ABB RobotStudio station: Palletixing_1.rspag

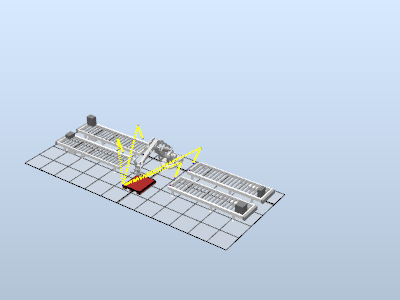
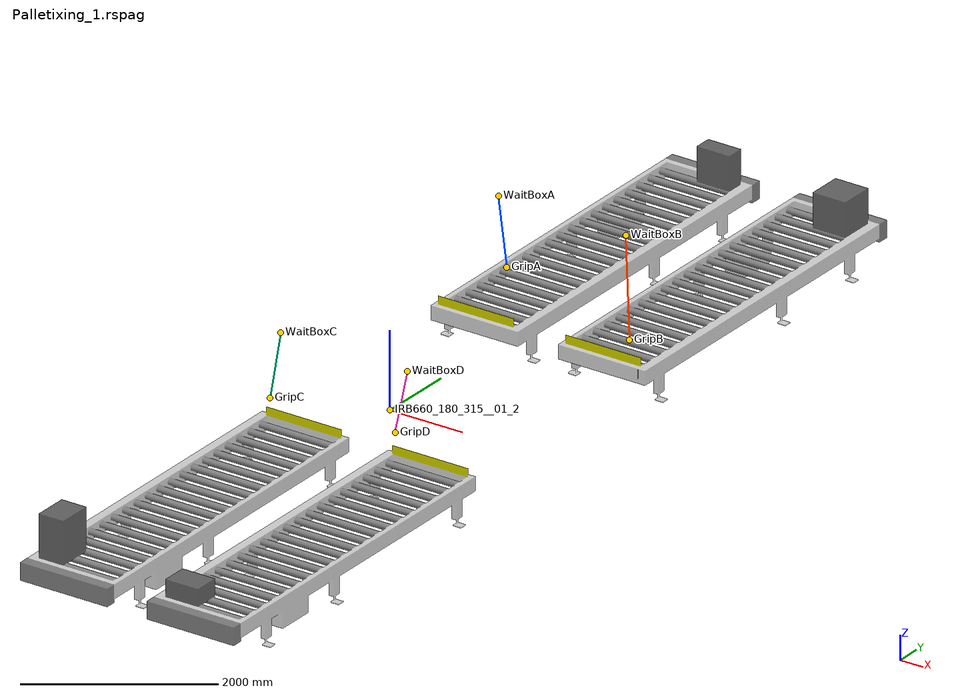
[picture v1: parts stored in the station drawn from their meshes, with robot base, taught points and paths (robot models come from the ABB library and are not in the file)]
--- station ---
Station Palletixing (saved by RobotStudio 22.3.10098.0)
Controller Controller2
  mechanical unit ROB_1: IRB660_180_315__01_2, 6 joints, base frame (0, 0, 0) mm
Layout (positions relative to the parent item):
  - IRB660_180_315__01_2 [mechanism, from Robots\IRB660_180_315__01.rslib] at (0, 0, 0) mm; joint values [0.1264, 0.8087, 0.1407, 0.1264] (rad or m)
  - Pallet1 [graphiccomponentgroup, from test\Pallet1.rslib] at (1000, 840, 377.87) mm, rotated rx 0 ry 0 rz 180 deg
    - MainBody [part, from test\Pallet1.rslib] at (-1900.1, 384.24, -377.87) mm
  - SC_InFeederA [smart component] at (435, 5540, 435) mm, rotated rx 0 ry 0 rz 180 deg
      signals: DI diNewBox, DO doBoxInPos, DI DiSizeBox
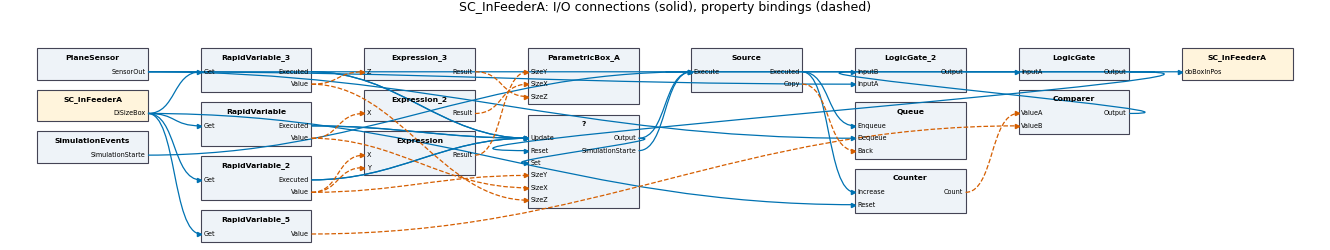
      connections:
        Source.Executed -> Queue.Enqueue
        PlaneSensor.SensorOut -> Queue.Dequeue
        PlaneSensor.SensorOut -> SC_InFeederA.doBoxInPos
        RapidVariable_3.Executed -> ?.Update
        RapidVariable.Executed -> ?.Update
        RapidVariable_2.Executed -> ?.Update
        RapidVariable_2.Executed -> ?.Update
        RapidVariable.Executed -> ?.Update
        RapidVariable_3.Executed -> ?.Update
        LogicGate.Output -> ?.Reset
        ?.Output -> ?.Set
        ?.Output -> Source.Execute
        LogicGate.Output -> Source.Execute
        ?.SimulationStarted -> Source.Execute
        SC_InFeederA.DiSizeBox -> RapidVariable.Get
        SC_InFeederA.DiSizeBox -> RapidVariable_2.Get
        SC_InFeederA.DiSizeBox -> RapidVariable_3.Get
        Source.Executed -> Counter.Increase
        SC_InFeederA.DiSizeBox -> Counter.Reset
        SC_InFeederA.DiSizeBox -> RapidVariable_5.Get
        Comparer.Output -> LogicGate_2.InputB
        PlaneSensor.SensorOut -> LogicGate_2.InputA
        LogicGate_2.Output -> LogicGate.InputA
        SimulationEvents.SimulationStarted -> Source.Execute
        Source.Copy => Queue.Back
        RapidVariable_2.Value => ?.SizeY
        RapidVariable.Value => ?.SizeX
        RapidVariable_3.Value => ?.SizeZ
        RapidVariable_2.Value => Expression.X
        Expression.Result => ParametricBox_A.SizeY
        RapidVariable_2.Value => Expression.Y
        RapidVariable.Value => Expression_2.X
        Expression_2.Result => ParametricBox_A.SizeX
        RapidVariable_3.Value => Expression_3.Z
        Expression_3.Result => ParametricBox_A.SizeZ
        Counter.Count => Comparer.ValueA
        RapidVariable_5.Value => Comparer.ValueB
    - InFeeder [part] at (435, 5140, -435) mm, rotated rx 0 ry 0 rz -90 deg, size 4244 x 1170 x 435 mm
    - Source [smart component, from Components\Source.rslib] at (435, 5140, -435) mm, rotated rx 0 ry 0 rz -90 deg
        properties: Source=ParametricBox_A; Copy=(none); Parent=(none); Position=[0 0 0]; Orientation=[0 0 0]; Transient=false; PhysicsBehavior=0
    - LinearMover [smart component, from Components\LinearMover.rslib] at (435, 5140, -435) mm, rotated rx 0 ry 0 rz -90 deg
        properties: Object=Queue; Direction=[0 -0.001 0]; Speed=0.5; Reference=Global; ReferenceObject=(none)
    - Queue [smart component, from Components\Queue.rslib] at (435, 5140, -435) mm, rotated rx 0 ry 0 rz -90 deg
        properties: Back=(none); Front=(none); Queue={59879bf6-beb7-4268-bf3d-d6b0f704d22e};{a24a8717-e6c1-41ba-83c6-47f9be62e9e9};{854ca087-3c3d-4bb9-8d85-1c4b9bd83209};{1b7bae8e-10d1-4233-8256-d01e01c4a4cd};{8b5e5753-a75c-4601-ac7b-2d1df5f60358};{555c76b8-d164-4f4a-8269-127b382f5ce1};{8e647ec2-27b4-49a6-b429-74ab6e4790a4};{bdffc5f9-98b3-472a-9b0a-d6f4ba94105b};{8ef266fb-d475-4d00-bda9-0d220e1673af};{4eefa4cf-f64c-4264-96e3-88afc0ee2385};{0a442b4f-4d82-4973-92c9-af11481ecd4b};{7e85bc6f-bf0a-45fb-b566-82c199c30cc5};{1e987258-a426-4c2d-bbfe-0a356d6c681f};{604d029a-7132-4a6c-8aca-46d3bcc26c59};{80aa472b-6015-4f67-8128-1b262151326c};{c680c479-d4ae-4059-8bb3-b634f61bb5f6};{a8d856c6-9330-41a9-ad49-869061775e72}; NumberOfObjects=1
    - PlaneSensor [smart component, from Components\PlaneSensor.rslib] at (435, 5140, -435) mm, rotated rx 0 ry 0 rz -90 deg
        properties: Origin=[1.14 0.485 0.435]; Axis1=[0 0 0.1]; Axis2=[0 -0.93 0]; SensedPart=(none)
      - _sensorPart_ [part], size 0 x 930 x 100 mm
    - LogicGate [smart component, from Components\LogicGate.rslib] at (435, 5140, -435) mm, rotated rx 0 ry 0 rz -90 deg
        properties: Operator=NOT; Delay=0
    - RapidVariable [smart component, from Components\RapidVariable.rslib] at (435, 5140, -435) mm, rotated rx 0 ry 0 rz -90 deg
        properties: DataType=num; Controller=Controller2; Task=T_ROB1; Module=Module1; Variable=widthBox; Value=400
    - RapidVariable_2 [smart component, from Components\RapidVariable.rslib] at (435, 5140, -435) mm, rotated rx 0 ry 0 rz -90 deg
        properties: DataType=num; Controller=Controller2; Task=T_ROB1; Module=Module1; Variable=depthBox; Value=200
    - RapidVariable_3 [smart component, from Components\RapidVariable.rslib] at (435, 5140, -435) mm, rotated rx 0 ry 0 rz -90 deg
        properties: DataType=num; Controller=Controller2; Task=T_ROB1; Module=Module1; Variable=heightBox; Value=400
    - ParametricBox_A [smart component, from Components\ParametricBox.rslib]
        properties: SizeX=0.4; SizeY=0.2; SizeZ=0.4; GeneratedPart=GeneratedPart; KeepGeometry=true
      - GeneratedPart [part], size 400 x 200 x 400 mm
    - Expression [smart component, from Components\Expression.rslib]
        properties: Expression=Y/1000; Result=0.2; Y=200
    - Expression_2 [smart component, from Components\Expression.rslib]
        properties: Expression=X/1000; Result=0.4; X=400
    - Expression_3 [smart component, from Components\Expression.rslib]
        properties: Expression=Z/1000; Result=0.4; Z=400
    - LogicGate_2 [smart component, from Components\LogicGate.rslib]
        properties: Operator=OR; Delay=0
    - RapidVariable_4 [smart component, from Components\RapidVariable.rslib]
        properties: DataType=num; Controller=(none); Task=; Module=; Variable=; Value=0
    - Comparer [smart component, from Components\Comparer.rslib]
        properties: ValueA=0; Operator=>=; ValueB=2
    - Counter [smart component, from Components\Counter.rslib]
        properties: Count=0
    - RapidVariable_5 [smart component, from Components\RapidVariable.rslib]
        properties: DataType=num; Controller=Controller2; Task=T_ROB1; Module=Module1; Variable=N; Value=2
    - SimulationEvents [smart component, from Components\SimulationEvents.rslib]
  - SC_InFeederC [smart component] at (-435, -5540, 435) mm
      signals: DI diNewBox, DO doBoxInPos, DI DiSizeBox
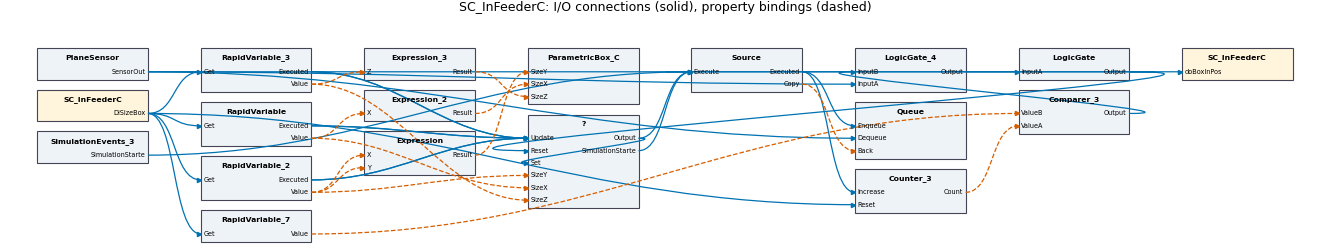
      connections:
        Source.Executed -> Queue.Enqueue
        PlaneSensor.SensorOut -> Queue.Dequeue
        PlaneSensor.SensorOut -> SC_InFeederC.doBoxInPos
        RapidVariable_3.Executed -> ?.Update
        RapidVariable.Executed -> ?.Update
        RapidVariable_2.Executed -> ?.Update
        RapidVariable_2.Executed -> ?.Update
        RapidVariable.Executed -> ?.Update
        RapidVariable_3.Executed -> ?.Update
        LogicGate.Output -> ?.Reset
        ?.Output -> ?.Set
        ?.Output -> Source.Execute
        LogicGate.Output -> Source.Execute
        ?.SimulationStarted -> Source.Execute
        SC_InFeederC.DiSizeBox -> RapidVariable.Get
        SC_InFeederC.DiSizeBox -> RapidVariable_2.Get
        SC_InFeederC.DiSizeBox -> RapidVariable_3.Get
        Source.Executed -> Counter_3.Increase
        SC_InFeederC.DiSizeBox -> Counter_3.Reset
        SC_InFeederC.DiSizeBox -> RapidVariable_7.Get
        Comparer_3.Output -> LogicGate_4.InputB
        PlaneSensor.SensorOut -> LogicGate_4.InputA
        LogicGate_4.Output -> LogicGate.InputA
        SimulationEvents_3.SimulationStarted -> Source.Execute
        Source.Copy => Queue.Back
        RapidVariable_2.Value => ?.SizeY
        RapidVariable.Value => ?.SizeX
        RapidVariable_3.Value => ?.SizeZ
        RapidVariable_2.Value => Expression.X
        Expression.Result => ParametricBox_C.SizeY
        RapidVariable_2.Value => Expression.Y
        RapidVariable.Value => Expression_2.X
        Expression_2.Result => ParametricBox_C.SizeX
        RapidVariable_3.Value => Expression_3.Z
        Expression_3.Result => ParametricBox_C.SizeZ
        RapidVariable_7.Value => Comparer_3.ValueB
        Counter_3.Count => Comparer_3.ValueA
    - InFeeder [part] at (435, 5140, -435) mm, rotated rx 0 ry 0 rz -90 deg, size 4244 x 1170 x 435 mm
    - Source [smart component, from Components\Source.rslib] at (435, 5140, -435) mm, rotated rx 0 ry 0 rz -90 deg
        properties: Source=ParametricBox_C; Copy=(none); Parent=(none); Position=[0 0 0]; Orientation=[0 0 0]; Transient=false; PhysicsBehavior=0
    - LinearMover [smart component, from Components\LinearMover.rslib] at (435, 5140, -435) mm, rotated rx 0 ry 0 rz -90 deg
        properties: Object=Queue; Direction=[0 0.001 0]; Speed=0.5; Reference=Global; ReferenceObject=(none)
    - Queue [smart component, from Components\Queue.rslib] at (435, 5140, -435) mm, rotated rx 0 ry 0 rz -90 deg
        properties: Back=(none); Front=(none); Queue={52c6f6fb-74d9-44ed-a61e-96cf36c5bd4c};{25b1f6b6-f2d7-4ebe-8c01-6ac80f9ece5e};{8c10390d-b4f7-40fa-a498-ef1ef82e99d7};{48a7697f-b334-4fe6-992c-7300ee66643c};{debe55c4-54e9-4823-967d-b62655e370e4};{01f9241d-2ba9-4314-a10c-5aca6cad913a};{541e0615-89a0-48f1-b9dd-00a0e8aaf4d0};{66341ac0-b4d0-470c-8dee-fd7ce2d6e368};{5d3dd006-543b-44f6-8dd8-8f7b57ebc5b3};{7561e20a-8e69-4836-96de-3675fc43be4e}; NumberOfObjects=0
    - PlaneSensor [smart component, from Components\PlaneSensor.rslib] at (435, 5140, -435) mm, rotated rx 0 ry 0 rz -90 deg
        properties: Origin=[1.14 0.485 0.435]; Axis1=[0 0 0.1]; Axis2=[0 -0.93 0]; SensedPart=(none)
      - _sensorPart_ [part], size 0 x 930 x 100 mm
    - LogicGate [smart component, from Components\LogicGate.rslib] at (435, 5140, -435) mm, rotated rx 0 ry 0 rz -90 deg
        properties: Operator=NOT; Delay=0
    - RapidVariable [smart component, from Components\RapidVariable.rslib] at (435, 5140, -435) mm, rotated rx 0 ry 0 rz -90 deg
        properties: DataType=num; Controller=Controller2; Task=T_ROB1; Module=Module1; Variable=widthBox; Value=300
    - RapidVariable_2 [smart component, from Components\RapidVariable.rslib] at (435, 5140, -435) mm, rotated rx 0 ry 0 rz -90 deg
        properties: DataType=num; Controller=Controller2; Task=T_ROB1; Module=Module1; Variable=depthBox; Value=400
    - RapidVariable_3 [smart component, from Components\RapidVariable.rslib] at (435, 5140, -435) mm, rotated rx 0 ry 0 rz -90 deg
        properties: DataType=num; Controller=Controller2; Task=T_ROB1; Module=Module1; Variable=heightBox; Value=500
    - ParametricBox_C [smart component, from Components\ParametricBox.rslib]
        properties: SizeX=0.3; SizeY=0.4; SizeZ=0.5; GeneratedPart=GeneratedPart; KeepGeometry=true
      - GeneratedPart [part], size 300 x 400 x 500 mm
    - Expression [smart component, from Components\Expression.rslib]
        properties: Expression=Y/1000; Result=0.4; Y=400
    - Expression_2 [smart component, from Components\Expression.rslib]
        properties: Expression=X/1000; Result=0.3; X=300
    - Expression_3 [smart component, from Components\Expression.rslib]
        properties: Expression=Z/1000; Result=0.5; Z=500
    - LogicGate_4 [smart component, from Components\LogicGate.rslib]
        properties: Operator=OR; Delay=0
    - Comparer_3 [smart component, from Components\Comparer.rslib]
        properties: ValueA=0; Operator=>=; ValueB=2
    - Counter_3 [smart component, from Components\Counter.rslib]
        properties: Count=0
    - RapidVariable_7 [smart component, from Components\RapidVariable.rslib]
        properties: DataType=num; Controller=Controller2; Task=T_ROB1; Module=Module1; Variable=N; Value=2
    - SimulationEvents_3 [smart component, from Components\SimulationEvents.rslib]
  - SC_InFeederD [smart component] at (1120, -5540, 435) mm
      signals: DI diNewBox, DO doBoxInPos, DI DiSizeBox
      connections:
        Source.Executed -> Queue.Enqueue
        PlaneSensor.SensorOut -> Queue.Dequeue
        PlaneSensor.SensorOut -> SC_InFeederD.doBoxInPos
        RapidVariable_3.Executed -> ?.Update
        RapidVariable.Executed -> ?.Update
        RapidVariable_2.Executed -> ?.Update
        RapidVariable_2.Executed -> ?.Update
        RapidVariable.Executed -> ?.Update
        RapidVariable_3.Executed -> ?.Update
        LogicGate.Output -> ?.Reset
        ?.Output -> ?.Set
        ?.Output -> Source.Execute
        LogicGate.Output -> Source.Execute
        ?.SimulationStarted -> Source.Execute
        SC_InFeederD.DiSizeBox -> RapidVariable.Get
        SC_InFeederD.DiSizeBox -> RapidVariable_2.Get
        SC_InFeederD.DiSizeBox -> RapidVariable_3.Get
        Source.Executed -> Counter_4.Increase
        SC_InFeederD.DiSizeBox -> RapidVariable_8.Get
        Comparer_4.Output -> LogicGate_5.InputB
        PlaneSensor.SensorOut -> LogicGate_5.InputA
        LogicGate_5.Output -> LogicGate.InputA
        SC_InFeederD.DiSizeBox -> Counter_4.Reset
        SimulationEvents_4.SimulationStarted -> Source.Execute
        Source.Copy => Queue.Back
        RapidVariable_2.Value => ?.SizeY
        RapidVariable.Value => ?.SizeX
        RapidVariable_3.Value => ?.SizeZ
        RapidVariable_2.Value => Expression.X
        Expression.Result => ParametricBox_D.SizeY
        RapidVariable_2.Value => Expression.Y
        RapidVariable.Value => Expression_2.X
        Expression_2.Result => ParametricBox_D.SizeX
        RapidVariable_3.Value => Expression_3.Z
        Expression_3.Result => ParametricBox_D.SizeZ
        Counter_4.Count => Comparer_4.ValueA
        RapidVariable_8.Value => Comparer_4.ValueB
    - InFeeder [part] at (435, 5140, -435) mm, rotated rx 0 ry 0 rz -90 deg, size 4244 x 1170 x 435 mm
    - Source [smart component, from Components\Source.rslib] at (435, 5140, -435) mm, rotated rx 0 ry 0 rz -90 deg
        properties: Source=ParametricBox_D; Copy=(none); Parent=(none); Position=[0 0 0]; Orientation=[0 0 0]; Transient=false; PhysicsBehavior=0
    - LinearMover [smart component, from Components\LinearMover.rslib] at (435, 5140, -435) mm, rotated rx 0 ry 0 rz -90 deg
        properties: Object=Queue; Direction=[0 0.001 0]; Speed=0.5; Reference=Global; ReferenceObject=(none)
    - Queue [smart component, from Components\Queue.rslib] at (435, 5140, -435) mm, rotated rx 0 ry 0 rz -90 deg
        properties: Back=(none); Front=(none); Queue={887726ed-16c2-49df-ba88-e57ece962b63};{8b0dd83f-e53a-43ce-833b-fe89e3d55376};{156f9ba2-dddb-422f-b2c1-abe5a9bc4498};{d9331796-f0d1-484d-ab00-a0cc222db9b9};{e1560b68-0188-4b83-ad28-061b1729fa91};{8e872459-965e-4969-a164-cafe7a149e64};{cc9c5c90-3e8b-4c06-9c9f-4edd16dc97a9};{0d97821e-1417-4d7a-8b3d-6921626bfc08};{88d902ee-d6c7-4e28-9c0e-ba93e6620a56};{51ea5b21-2d51-4a57-9619-941efac5c7e2};{364fce12-9345-48be-9ecb-459c9ffcb072};{c2a1d569-b57c-49d8-ad33-5409f4edd47a}; NumberOfObjects=0
    - PlaneSensor [smart component, from Components\PlaneSensor.rslib] at (435, 5140, -435) mm, rotated rx 0 ry 0 rz -90 deg
        properties: Origin=[1.14 0.485 0.435]; Axis1=[0 0 0.1]; Axis2=[0 -0.93 0]; SensedPart=(none)
      - _sensorPart_ [part], size 0 x 930 x 100 mm
    - LogicGate [smart component, from Components\LogicGate.rslib] at (435, 5140, -435) mm, rotated rx 0 ry 0 rz -90 deg
        properties: Operator=NOT; Delay=0
    - RapidVariable [smart component, from Components\RapidVariable.rslib] at (435, 5140, -435) mm, rotated rx 0 ry 0 rz -90 deg
        properties: DataType=num; Controller=Controller2; Task=T_ROB1; Module=Module1; Variable=widthBox; Value=400
    - RapidVariable_2 [smart component, from Components\RapidVariable.rslib] at (435, 5140, -435) mm, rotated rx 0 ry 0 rz -90 deg
        properties: DataType=num; Controller=Controller2; Task=T_ROB1; Module=Module1; Variable=depthBox; Value=300
    - RapidVariable_3 [smart component, from Components\RapidVariable.rslib] at (435, 5140, -435) mm, rotated rx 0 ry 0 rz -90 deg
        properties: DataType=num; Controller=Controller2; Task=T_ROB1; Module=Module1; Variable=heightBox; Value=200
    - ParametricBox_D [smart component, from Components\ParametricBox.rslib]
        properties: SizeX=0.4; SizeY=0.3; SizeZ=0.2; GeneratedPart=GeneratedPart; KeepGeometry=true
      - GeneratedPart [part], size 400 x 300 x 200 mm
    - Expression [smart component, from Components\Expression.rslib]
        properties: Expression=Y/1000; Result=0.3; Y=300
    - Expression_2 [smart component, from Components\Expression.rslib]
        properties: Expression=X/1000; Result=0.4; X=400
    - Expression_3 [smart component, from Components\Expression.rslib]
        properties: Expression=Z/1000; Result=0.2; Z=200
    - RapidVariable_8 [smart component, from Components\RapidVariable.rslib]
        properties: DataType=num; Controller=Controller2; Task=T_ROB1; Module=Module1; Variable=N; Value=3
    - Counter_4 [smart component, from Components\Counter.rslib]
        properties: Count=0
    - Comparer_4 [smart component, from Components\Comparer.rslib]
        properties: ValueA=0; Operator=>=; ValueB=3
    - LogicGate_5 [smart component, from Components\LogicGate.rslib]
        properties: Operator=OR; Delay=0
    - SimulationEvents_4 [smart component, from Components\SimulationEvents.rslib]
  - SC_InFeederB [smart component] at (2000, 5540, 435) mm, rotated rx 0 ry 0 rz 180 deg
      signals: DI diNewBox, DO doBoxInPos, DI DiSizeBox
      connections:
        Source.Executed -> Queue.Enqueue
        PlaneSensor.SensorOut -> Queue.Dequeue
        PlaneSensor.SensorOut -> SC_InFeederB.doBoxInPos
        RapidVariable_3.Executed -> ?.Update
        RapidVariable.Executed -> ?.Update
        RapidVariable_2.Executed -> ?.Update
        RapidVariable_2.Executed -> ?.Update
        RapidVariable.Executed -> ?.Update
        RapidVariable_3.Executed -> ?.Update
        LogicGate.Output -> ?.Reset
        ?.Output -> ?.Set
        ?.Output -> Source.Execute
        LogicGate.Output -> Source.Execute
        ?.SimulationStarted -> Source.Execute
        SC_InFeederB.DiSizeBox -> RapidVariable.Get
        SC_InFeederB.DiSizeBox -> RapidVariable_2.Get
        SC_InFeederB.DiSizeBox -> RapidVariable_3.Get
        Source.Executed -> Counter_2.Increase
        SC_InFeederB.DiSizeBox -> Counter_2.Reset
        SC_InFeederB.DiSizeBox -> RapidVariable_6.Get
        Comparer_2.Output -> LogicGate_3.InputB
        PlaneSensor.SensorOut -> LogicGate_3.InputA
        LogicGate_3.Output -> LogicGate.InputA
        SimulationEvents_2.SimulationStarted -> Source.Execute
        Source.Copy => Queue.Back
        RapidVariable_2.Value => ?.SizeY
        RapidVariable.Value => ?.SizeX
        RapidVariable_3.Value => ?.SizeZ
        RapidVariable_2.Value => Expression.X
        Expression.Result => ParametricBox_B.SizeY
        RapidVariable_2.Value => Expression.Y
        RapidVariable.Value => Expression_2.X
        Expression_2.Result => ParametricBox_B.SizeX
        RapidVariable_3.Value => Expression_3.Z
        Expression_3.Result => ParametricBox_B.SizeZ
        Counter_2.Count => Comparer_2.ValueA
        RapidVariable_6.Value => Comparer_2.ValueB
    - InFeeder [part] at (435, 5140, -435) mm, rotated rx 0 ry 0 rz -90 deg, size 4244 x 1170 x 435 mm
    - Source [smart component, from Components\Source.rslib] at (435, 5140, -435) mm, rotated rx 0 ry 0 rz -90 deg
        properties: Source=ParametricBox_B; Copy=(none); Parent=(none); Position=[0 0 0]; Orientation=[0 0 0]; Transient=false; PhysicsBehavior=0
    - LinearMover [smart component, from Components\LinearMover.rslib] at (435, 5140, -435) mm, rotated rx 0 ry 0 rz -90 deg
        properties: Object=Queue; Direction=[0 -0.001 0]; Speed=0.5; Reference=Global; ReferenceObject=(none)
    - Queue [smart component, from Components\Queue.rslib] at (435, 5140, -435) mm, rotated rx 0 ry 0 rz -90 deg
        properties: Back=(none); Front=(none); Queue={e0fa0a83-854e-4275-bcb0-fbd7c086035f};{272aca57-2305-423f-b320-0d412a35e15d};{52ac2ab8-f7a7-4606-8d1f-cf022a095ca7};{99a9a24d-aa25-48da-a172-038a36b4bb77};{9b0f4713-29e7-4eca-8b68-f50dc9cad909};{3cfba3e1-b737-4f56-b0eb-bcaad8e71801};{4216f030-429a-4b76-9731-3bf365c2aa94};{92b21d38-edd2-4a8f-9b58-f375044d3cec};{fac17516-3dfd-4b60-bf8b-2b1232ffe8fe};{7d8e88de-14e2-4d50-a1ca-70d82d6d6da5};{1db5e097-2bbb-4e32-821e-b7323cd4b91f};{3c734a2e-fdf5-43d4-ace7-3793a3cfd0f2};{b64fa727-8d83-43cf-b826-b906ec598db5};{7716e356-0133-4851-92b4-e3b64b98599a};{3ca38520-0a75-41a6-b88a-40c77d9361a7};{304ac827-ded2-41a3-a0bd-cc434ea2ca2e};{8f60f646-6345-40a9-a12a-a4b380d49997}; NumberOfObjects=0
    - PlaneSensor [smart component, from Components\PlaneSensor.rslib] at (435, 5140, -435) mm, rotated rx 0 ry 0 rz -90 deg
        properties: Origin=[1.14 0.485 0.435]; Axis1=[0 0 0.1]; Axis2=[0 -0.93 0]; SensedPart=(none)
      - _sensorPart_ [part], size 0 x 930 x 100 mm
    - LogicGate [smart component, from Components\LogicGate.rslib] at (435, 5140, -435) mm, rotated rx 0 ry 0 rz -90 deg
        properties: Operator=NOT; Delay=0
    - RapidVariable [smart component, from Components\RapidVariable.rslib] at (435, 5140, -435) mm, rotated rx 0 ry 0 rz -90 deg
        properties: DataType=num; Controller=Controller2; Task=T_ROB1; Module=Module1; Variable=widthBox; Value=400
    - RapidVariable_2 [smart component, from Components\RapidVariable.rslib] at (435, 5140, -435) mm, rotated rx 0 ry 0 rz -90 deg
        properties: DataType=num; Controller=Controller2; Task=T_ROB1; Module=Module1; Variable=depthBox; Value=400
    - RapidVariable_3 [smart component, from Components\RapidVariable.rslib] at (435, 5140, -435) mm, rotated rx 0 ry 0 rz -90 deg
        properties: DataType=num; Controller=Controller2; Task=T_ROB1; Module=Module1; Variable=heightBox; Value=400
    - ParametricBox_B [smart component, from Components\ParametricBox.rslib]
        properties: SizeX=0.4; SizeY=0.4; SizeZ=0.4; GeneratedPart=GeneratedPart; KeepGeometry=true
      - GeneratedPart [part], size 400 x 400 x 400 mm
    - Expression [smart component, from Components\Expression.rslib]
        properties: Expression=Y/1000; Result=0.4; Y=400
    - Expression_2 [smart component, from Components\Expression.rslib]
        properties: Expression=X/1000; Result=0.4; X=400
    - Expression_3 [smart component, from Components\Expression.rslib]
        properties: Expression=Z/1000; Result=0.4; Z=400
    - RapidVariable_6 [smart component, from Components\RapidVariable.rslib]
        properties: DataType=num; Controller=Controller2; Task=T_ROB1; Module=Module1; Variable=N; Value=2
    - Counter_2 [smart component, from Components\Counter.rslib]
        properties: Count=0
    - Comparer_2 [smart component, from Components\Comparer.rslib]
        properties: ValueA=0; Operator=>=; ValueB=2
    - LogicGate_3 [smart component, from Components\LogicGate.rslib]
        properties: Operator=OR; Delay=0
    - SimulationEvents_2 [smart component, from Components\SimulationEvents.rslib]
  -  SC_VacuumGripper [smart component] at (2800.1, 355.76, 1247.5) mm, rotated rx 180 ry 0 rz 180 deg
      properties: PartInGripper=(none); SavedState.vacuum_gripper=<ProjectState name="vacuum_gripper" description="" date="2022-07-14T11:56:36.5223942+07:00">
  <ObjectStates>
    <StandardState objectId="{b8ed2f7f-5b48-42f8-af5a-16fdca5917d1}">
      <Transform matrix="[[-1 0 0 0] [0 1 0 0] [0 0 -1 0] [1.91 2.18919440951939E-15 1.833 1]]" />
      <AttachmentParent parentId="{0d465377-8a6a-4130-92d5-134fd99cc6ca}" matrix="[[-1 0 0 0] [0 1 0 0] [0 0 -1 0] [1.91 0 1.833 1]]" />
      <Visible value="True" />
      <DynamicProperty name="PartInGripper" value="" />
      <IOSignal name="diAttach" value="0" />
      <IOSignal name="doAttached" value="0" />
      <IOSignal name="doDetached" value="1" />
    </StandardState>
    <StandardState objectId="{19b66e55-08e3-4c2f-9ed3-921632e336bf}">
      <Transform matrix="[[1 0 0 0] [0 1 0 0] [0 0 1 0] [0 0 0 1]]" />
      <AttachmentParent parentId="" matrix="" />
      <Visible value="True" />
    </StandardState>
    <StandardState objectId="{3783844f-07c0-4e1d-93e4-a36a9a4f0c9b}">
      <Transform matrix="[[1 0 0 0] [0 1 0 0] [0 0 1 0] [0 0 0 1]]" />
      <AttachmentParent parentId="" matrix="" />
      <Visible value="True" />
      <DynamicProperty name="Start" value="[0 0 0.15]" />
      <DynamicProperty name="End" value="[0 0 0.25]" />
      <DynamicProperty name="Radius" value="0.001" />
      <DynamicProperty name="SensedPart" value="" />
      <DynamicProperty name="SensedPoint" value="[0 0 0]" />
      <IOSignal name="Active" value="0" />
      <IOSignal name="SensorOut" value="0" />
    </StandardState>
    <StandardState objectId="{d4abe88d-1c90-474c-8fb7-a108e99152a3}">
      <Transform matrix="[[1 0 0 0] [0 1 0 0] [0 0 1 0] [0 0 0 1]]" />
      <AttachmentParent parentId="" matrix="" />
      <Visible value="True" />
      <DynamicProperty name="Parent" value="{19b66e55-08e3-4c2f-9ed3-921632e336bf}" />
      <DynamicProperty name="Flange" value="0" />
      <DynamicProperty name="Child" value="" />
      <DynamicProperty name="Mount" value="False" />
      <DynamicProperty name="Offset" value="[0 0 0]" />
      <DynamicProperty name="Orientation" value="[0 0 0]" />
      <IOSignal name="Execute" value="0" />
      <IOSignal name="Executed" value="0" />
    </StandardState>
    <StandardState objectId="{040f266f-09a0-41e9-ad9d-4da25baf776e}">
      <Transform matrix="[[1 0 0 0] [0 1 0 0] [0 0 1 0] [0 0 0 1]]" />
      <AttachmentParent parentId="" matrix="" />
      <Visible value="True" />
      <DynamicProperty name="Child" value="" />
      <DynamicProperty name="KeepPosition" value="True" />
      <IOSignal name="Execute" value="0" />
      <IOSignal name="Executed" value="0" />
    </StandardState>
    <StandardState objectId="{678b1997-4bb7-41a8-beb4-cc493f3f5a97}">
      <Transform matrix="[[1 0 0 0] [0 1 0 0] [0 0 1 0] [0 0 0 1]]" />
      <AttachmentParent parentId="" matrix="" />
      <Visible value="True" />
      <DynamicProperty name="Operator" value="NOT" />
      <DynamicProperty name="Delay" value="0" />
      <IOSignal name="InputA" value="0" />
      <IOSignal name="InputB" value="0" />
      <IOSignal name="Output" value="1" />
    </StandardState>
    <StandardState objectId="{483069c4-b9ae-477b-8e71-91e4b5074d60}">
      <Transform matrix="[[1 0 0 0] [0 1 0 0] [0 0 1 0] [0 0 0 1]]" />
      <AttachmentParent parentId="" matrix="" />
      <Visible value="True" />
      <IOSignal name="Set" value="0" />
      <IOSignal name="Reset" value="0" />
      <IOSignal name="Output" value="0" />
      <IOSignal name="InvOutput" value="1" />
    </StandardState>
    <StandardState objectId="{b662bc42-54f4-44d6-8bbf-b0fc7c07bb5b}">
      <PhysicsMotionControl value="None" />
      <Visible value="True" />
    </StandardState>
    <StandardState objectId="{6a989055-ac24-4bcf-b246-c249199d1956}">
      <Visible value="False" />
    </StandardState>
  </ObjectStates>
</ProjectState>; SavedStates=vacuum_gripper
      signals: DI diAttach, DO doAttached, DO doDetached, DI diAttachB, DI diAttachD, DI diAttachE, DO doAttachedB, DO doDetachedB, DO doAttachedD, DO doDetachedD, DO doAttachedE, DO doDetachedE
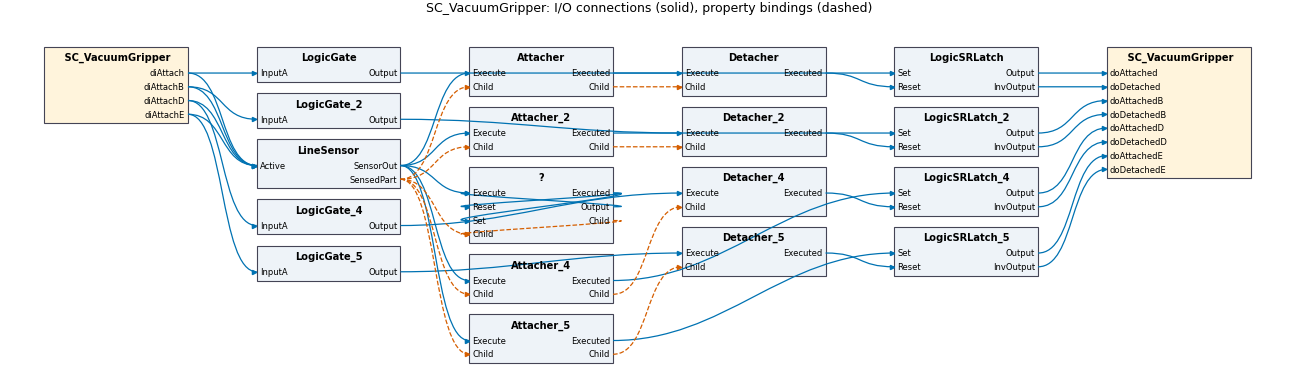
      connections:
         SC_VacuumGripper.diAttach -> LineSensor.Active
        LineSensor.SensorOut -> Attacher.Execute
         SC_VacuumGripper.diAttach -> LogicGate.InputA
        LogicGate.Output -> Detacher.Execute
        Attacher.Executed -> LogicSRLatch.Set
        Detacher.Executed -> LogicSRLatch.Reset
        LogicSRLatch.Output ->  SC_VacuumGripper.doAttached
        LogicSRLatch.InvOutput ->  SC_VacuumGripper.doDetached
        Attacher_2.Executed -> LogicSRLatch_2.Set
        Detacher_2.Executed -> LogicSRLatch_2.Reset
         SC_VacuumGripper.diAttachB -> LogicGate_2.InputA
        LineSensor.SensorOut -> Attacher_2.Execute
        LogicSRLatch_2.Output ->  SC_VacuumGripper.doAttachedB
        LogicSRLatch_2.InvOutput ->  SC_VacuumGripper.doDetachedB
        LogicGate_2.Output -> Detacher_2.Execute
        LineSensor.SensorOut -> ?.Execute
        ?.Executed -> ?.Reset
        ?.Executed -> ?.Set
         SC_VacuumGripper.diAttachB -> LineSensor.Active
        ?.Output -> ?.Execute
         SC_VacuumGripper.diAttachD -> LineSensor.Active
         SC_VacuumGripper.diAttachE -> LineSensor.Active
         SC_VacuumGripper.diAttachD -> LogicGate_4.InputA
        LogicGate_4.Output -> Detacher_4.Execute
        LineSensor.SensorOut -> Attacher_4.Execute
        Attacher_4.Executed -> LogicSRLatch_4.Set
        Detacher_4.Executed -> LogicSRLatch_4.Reset
        LogicSRLatch_4.Output ->  SC_VacuumGripper.doAttachedD
        LogicSRLatch_4.InvOutput ->  SC_VacuumGripper.doDetachedD
         SC_VacuumGripper.diAttachE -> LogicGate_5.InputA
        LineSensor.SensorOut -> Attacher_5.Execute
        Attacher_5.Executed -> LogicSRLatch_5.Set
        LogicGate_5.Output -> Detacher_5.Execute
        Detacher_5.Executed -> LogicSRLatch_5.Reset
        LogicSRLatch_5.Output ->  SC_VacuumGripper.doAttachedE
        LogicSRLatch_5.InvOutput ->  SC_VacuumGripper.doDetachedE
        LineSensor.SensedPart => Attacher.Child
        Attacher.Child => Detacher.Child
        LineSensor.SensedPart => Attacher_2.Child
        Attacher_2.Child => Detacher_2.Child
        LineSensor.SensedPart => ?.Child
        ?.Child => ?.Child
        LineSensor.SensedPart => Attacher_4.Child
        Attacher_4.Child => Detacher_4.Child
        LineSensor.SensedPart => Attacher_5.Child
        Attacher_5.Child => Detacher_5.Child
    - VacuumGripper [mechanism] at (0, 0, 0) mm
        TCP tGripper at (0, 0, 197.5) mm
        links: vacuum_gripper
    - LineSensor [smart component, from Components\LineSensor.rslib]
        properties: Start=[0 0 0.15]; End=[0 0 0.25]; Radius=0.005; SensedPart=(none); SensedPoint=[2.80010034179687 0.355763061523438 0.550052917480469]
      - _sensorPart_ [part], size 10 x 10 x 100 mm
    - Attacher [smart component, from Components\Attacher.rslib]
        properties: Parent=VacuumGripper; Flange=0; Child=(none); Mount=false; Offset=[0 0 0]; Orientation=[0 0 0]
    - Detacher [smart component, from Components\Detacher.rslib]
        properties: Child=(none); KeepPosition=true
    - LogicGate [smart component, from Components\LogicGate.rslib]
        properties: Operator=NOT; Delay=0
    - LogicSRLatch [smart component, from Components\LogicSRLatch.rslib]
    - Attacher_2 [smart component, from Components\Attacher.rslib]
        properties: Parent=VacuumGripper; Flange=0; Child=(none); Mount=false; Offset=[0 0 0]; Orientation=[0 0 0]
    - Detacher_2 [smart component, from Components\Detacher.rslib]
        properties: Child=(none); KeepPosition=true
    - LogicSRLatch_2 [smart component, from Components\LogicSRLatch.rslib]
    - LogicGate_2 [smart component, from Components\LogicGate.rslib]
        properties: Operator=NOT; Delay=0
    - Attacher_4 [smart component, from Components\Attacher.rslib]
        properties: Parent=(none); Flange=0; Child=(none); Mount=false; Offset=[0 0 0]; Orientation=[0 0 0]
    - Detacher_4 [smart component, from Components\Detacher.rslib]
        properties: Child=(none); KeepPosition=true
    - LogicGate_4 [smart component, from Components\LogicGate.rslib]
        properties: Operator=NOT; Delay=0
    - LogicSRLatch_4 [smart component, from Components\LogicSRLatch.rslib]
    - Attacher_5 [smart component, from Components\Attacher.rslib]
        properties: Parent=(none); Flange=0; Child=(none); Mount=false; Offset=[0 0 0]; Orientation=[0 0 0]
    - Detacher_5 [smart component, from Components\Detacher.rslib]
        properties: Child=(none); KeepPosition=true
    - LogicGate_5 [smart component, from Components\LogicGate.rslib]
        properties: Operator=NOT; Delay=0
    - LogicSRLatch_5 [smart component, from Components\LogicSRLatch.rslib]
Attachment: Workobject_BoxA is attached to InFeeder
Attachment: Workobject_BoxC is attached to InFeeder
Attachment: Workobject_BoxD is attached to InFeeder
Attachment: Workobject_BoxB is attached to InFeeder
Attachment:  SC_VacuumGripper is attached to IRB660_180_315__01_2 / Link6
Station logic (signal -> signal, property => property):
  Controller2.DoSizeBoxA -> SC_InFeederA.DiSizeBox
  Controller2.DoSizeBoxC -> SC_InFeederC.DiSizeBox
  Controller2.DoSizeBoxD -> SC_InFeederD.DiSizeBox
  SC_InFeederA.doBoxInPos -> Controller2.di_BoxInPosA
  SC_InFeederC.doBoxInPos -> Controller2.di_BoxInPosC
  SC_InFeederD.doBoxInPos -> Controller2.di_BoxInPosD
  Controller2.DoSizeBoxB -> SC_InFeederB.DiSizeBox
  SC_InFeederB.doBoxInPos -> Controller2.di_BoxInPosB
  LineSensor_3.SensorOut -> Attacher_A.Execute
  Controller2.do_DetachA -> Detacher_A.Execute
  Controller2.do_AttachA -> LineSensor_3.Active
  Controller2.do_AttachA ->  SC_VacuumGripper.diAttach
  Controller2.do_AttachB ->  SC_VacuumGripper.diAttachB
  Controller2.do_AttachC ->  SC_VacuumGripper.diAttachD
  Controller2.do_AttachD ->  SC_VacuumGripper.diAttachE
Targets, tools, work objects and paths stored in the station and not in the controller backup, written as RAPID:
! task T_ROB1
MODULE Module1
  PROC Path_10()
    MoveL Home,v1000,z100,tGripper\WObj:=wobj0;
    MoveL WaitBoxA,v1000,z100,tGripper\WObj:=Workobject_BoxA;
    MoveL WaitBoxB,v1000,z100,tGripper\WObj:=Workobject_BoxB;
    MoveJ WaitBoxC,v1000,z100,tGripper\WObj:=Workobject_BoxC;
    MoveL WaitBoxD,v1000,z100,tGripper\WObj:=Workobject_BoxD;
    MoveJ OffsetOnPallet,v1000,z100,tGripper\WObj:=Workobject_Pallet;
    MoveL Home,v1000,z100,tGripper\WObj:=wobj0;
    MoveL GripA,v1000,z100,tGripper\WObj:=Workobject_BoxA;
    MoveL GripB,v1000,z100,tGripper\WObj:=Workobject_BoxB;
    MoveJ GripC,v1000,z100,tGripper\WObj:=Workobject_BoxC;
    MoveL GripD,v1000,z100,tGripper\WObj:=Workobject_BoxD;
  ENDPROC
ENDMODULE


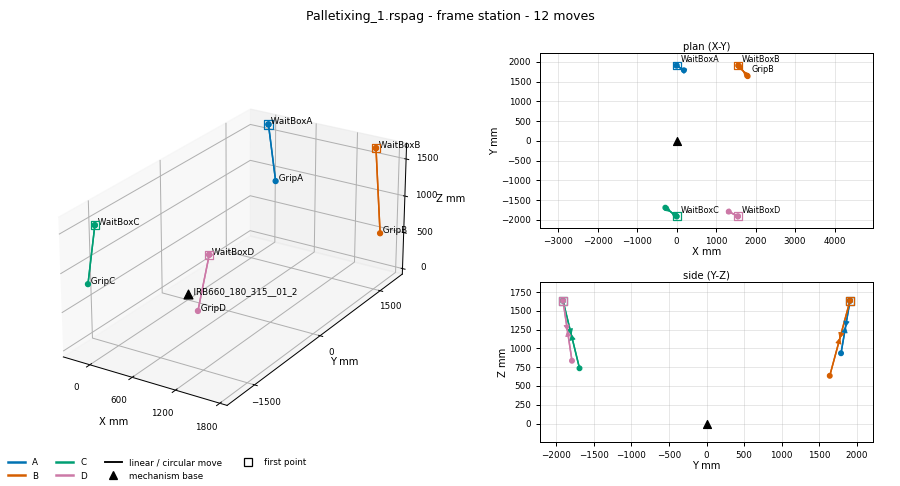
[picture p0: tool path of Palletixing_1.rspag in frame station, 12 of 24 moves have a stored position in this frame; points joined in program order, loops and branches not executed]
--- Backups/Controller2/RAPID/TASK1/PROGMOD/CalibData.mod ---
MODULE CalibData
    PERS tooldata tGripper:=[TRUE,[[0,0,197.500488281],[1,0,0,0]],[25,[0,0.001093272,116.889125016],[1,0,0,0],0,0,0]];
    TASK PERS wobjdata Workobject_BoxA:=[FALSE,TRUE,"",[[435,1540,435],[0.707106781,0,0,0.707106781]],[[0,0,0],[1,0,0,0]]];
    TASK PERS wobjdata Workobject_BoxB:=[FALSE,TRUE,"",[[2000,1540,435],[0.707106781,0,0,0.707106781]],[[0,0,0],[1,0,0,0]]];
    TASK PERS wobjdata Workobject_BoxC:=[FALSE,TRUE,"",[[-435,-1540,435],[0.707106781,0,0,-0.707106781]],[[0,0,0],[1,0,0,0]]];
    TASK PERS wobjdata Workobject_BoxD:=[FALSE,TRUE,"",[[1120,-1540,435],[0.707106781,0,0,-0.707106781]],[[0,0,0],[1,0,0,0]]];
    TASK PERS wobjdata Workobject_Pallet:=[FALSE,TRUE,"",[[2900.1,-544.237,150],[0.707106781,0,0,0.707106781]],[[0,0,0],[1,0,0,0]]];
ENDMODULE

--- Backups/Controller2/RAPID/TASK1/PROGMOD/Module1.mod ---
MODULE Module1
     PERS num widthBox;
     PERS num depthBox;
     PERS num heightBox;
     PERS num N;
     PERS num fittedBox;
    CONST robtarget Home:=[[1910,0,1833],[0,0,1,0],[0,0,0,0],[9E+09,9E+09,9E+09,9E+09,9E+09,9E+09]];
    CONST robtarget WaitBoxA:=[[370,435,1200.499511719],[0,0,1,0],[1,0,-1,0],[9E+09,9E+09,9E+09,9E+09,9E+09,9E+09]];
    CONST robtarget WaitBoxB:=[[370,435,1200.499511719],[0,0,1,0],[0,0,-1,0],[9E+09,9E+09,9E+09,9E+09,9E+09,9E+09]];
    CONST robtarget WaitBoxC:=[[370,435,1200.499511719],[0,0,1,0],[-2,0,0,0],[9E+09,9E+09,9E+09,9E+09,9E+09,9E+09]];
    CONST robtarget WaitBoxD:=[[370,435,1200.499511719],[0,0,1,0],[-1,0,0,0],[9E+09,9E+09,9E+09,9E+09,9E+09,9E+09]];

    PERS robtarget GripA:=[[250,250,500],[0,0,1,0],[0,0,-1,0],[9E+9,9E+9,9E+9,9E+9,9E+9,9E+9]];
    PERS robtarget GripB:=[[100,200,200],[0,0,1,0],[0,0,-1,0],[9E+9,9E+9,9E+9,9E+9,9E+9,9E+9]];
    PERS robtarget GripC:=[[150,150,300],[0,0,1,0],[-2,0,0,0],[9E+9,9E+9,9E+9,9E+9,9E+9,9E+9]];
    PERS robtarget GripD:=[[250,200,400],[0,0,1,0],[0,0,-1,0],[9E+9,9E+9,9E+9,9E+9,9E+9,9E+9]];
    PERS robtarget OffsetOnPallet:=[[800,600,1500],[0,0.707107,0.707107,0],[-1,0,-1,0],[9E+9,9E+9,9E+9,9E+9,9E+9,9E+9]];
    PERS robtarget BoxOnPallet:=[[800,600,1000],[0,0.707107,0.707107,0],[-1,0,-1,0],[9E+9,9E+9,9E+9,9E+9,9E+9,9E+9]];
    PERS pos tgPos{50};
    PERS pos offset{50};
    PERS num no{50};
    PERS num config{50};
    VAR bool repeat := TRUE;
    !***********************************************************
    !
    ! Module:  Module1
    !
    ! Description:
    !   <Insert description here>
    !
    ! Author: USER
    !
    ! Version: 1.0
    !
    !***********************************************************


    !***********************************************************
    !
    ! Procedure main
    !
    !   This is the entry point of your program
    !
    !***********************************************************
    PROC main()
        ConfJ\Off;
        ConfL\Off;
          WHILE repeat DO
               FOR i from 1 TO fittedBox DO
                    BoxOnPallet.trans := tgPos{i};
                    OffsetOnPallet.trans := offset{i};
                    IF no{i} = 1 THEN
                         A;
                    ELSEIF no{i} = 2 THEN
                         B;
                    ELSEIF no{i} = 3 THEN
                         C;
                    ELSEIF no{i} = 4 THEN
                         D;
                    endif
               ENDFOR
               repeat :=FALSE;
          ENDWHILE
          FOR i FROM 1 TO fittedBox DO
               tgPos{i} := [0,0,0];
               offset{i} := [0,0,0];
               no{i} := 0;
               N := 0;
               fittedBox := 0;
          ENDFOR

          repeat := TRUE;
    ENDPROC

    PROC A()
        MoveJ WaitBoxA,v1000,z100,tGripper\WObj:=Workobject_BoxA;
        WaitDI di_BoxInPosA,1;
        MoveL GripA,v1000,fine,tGripper\WObj:=Workobject_BoxA;
        SetDO do_AttachA,1;
        MoveL WaitBoxA,v1000,z100,tGripper\WObj:=Workobject_BoxA;
        MoveJ OffsetOnPallet,v1000,z100,tGripper\WObj:=Workobject_Pallet;
        MoveL BoxOnPallet,v1000,fine,tGripper\WObj:=Workobject_Pallet;
        SetDO do_AttachA,0;
        MoveL OffsetOnPallet,v1000,z100,tGripper\WObj:=Workobject_Pallet;
    ENDPROC

    PROC B()
        MoveJ WaitBoxB,v1000,z100,tGripper\WObj:=Workobject_BoxB;
        WaitDI di_BoxInPosB,1;
        MoveL GripB,v1000,fine,tGripper\WObj:=Workobject_BoxB;
        SetDO do_AttachB,1;
        MoveL WaitBoxB,v1000,z100,tGripper\WObj:=Workobject_BoxB;
        MoveJ OffsetOnPallet,v1000,z100,tGripper\WObj:=Workobject_Pallet;
        MoveL BoxOnPallet,v1000,fine,tGripper\WObj:=Workobject_Pallet;
        SetDO do_AttachB,0;
        MoveL OffsetOnPallet,v1000,z100,tGripper\WObj:=Workobject_Pallet;
    ENDPROC

    PROC C()
        MoveJ WaitBoxC,v1000,z100,tGripper\WObj:=Workobject_BoxC;
        WaitDI di_BoxInPosC,1;
        MoveL GripC,v1000,fine,tGripper\WObj:=Workobject_BoxC;
        SetDO do_AttachC,1;
        MoveL WaitBoxC,v1000,z100,tGripper\WObj:=Workobject_BoxC;
        MoveJ OffsetOnPallet,v1000,z100,tGripper\WObj:=Workobject_Pallet;
        MoveL BoxOnPallet,v1000,fine,tGripper\WObj:=Workobject_Pallet;
        SetDO do_AttachC,0;
        MoveL OffsetOnPallet,v1000,z100,tGripper\WObj:=Workobject_Pallet;
    ENDPROC

    PROC D()
        MoveJ WaitBoxD,v1000,z100,tGripper\WObj:=Workobject_BoxD;
        WaitDI di_BoxInPosD,1;
        MoveL GripD,v1000,fine,tGripper\WObj:=Workobject_BoxD;
        SetDO do_AttachD,1;
        MoveL WaitBoxD,v1000,z100,tGripper\WObj:=Workobject_BoxD;
        MoveJ OffsetOnPallet,v1000,z100,tGripper\WObj:=Workobject_Pallet;
        MoveL BoxOnPallet,v1000,fine,tGripper\WObj:=Workobject_Pallet;
        SetDO do_AttachD,0;
        MoveL OffsetOnPallet,v1000,z100,tGripper\WObj:=Workobject_Pallet;
    ENDPROC

ENDMODULE

--- Backups/Controller2/SYSPAR/EIO.cfg ---
EIO:CFG_1.0:6:1::
#
EIO_SIGNAL:

      -Name "DoSizeBoxA" -SignalType "DO" -Access "All"

      -Name "DoSizeBoxB" -SignalType "DO" -Access "All"

      -Name "DoSizeBoxC" -SignalType "DO" -Access "All"

      -Name "DoSizeBoxD" -SignalType "DO" -Access "All"

      -Name "do_AttachA" -SignalType "DO" -Access "All"

      -Name "do_AttachB" -SignalType "DO" -Access "All"

      -Name "do_AttachC" -SignalType "DO" -Access "All"

      -Name "do_AttachD" -SignalType "DO" -Access "All"

      -Name "di_BoxInPosA" -SignalType "DI" -Access "All"

      -Name "di_BoxInPosB" -SignalType "DI" -Access "All"

      -Name "di_BoxInPosC" -SignalType "DI" -Access "All"

      -Name "di_BoxInPosD" -SignalType "DI" -Access "All"

      -Name "do_DetachA" -SignalType "DO" -Access "All"
